// Mitsubishi GX Works2 project: Traffic light_MyTest   PLC: FX3U/FX3UC

PROGRAM MAIN
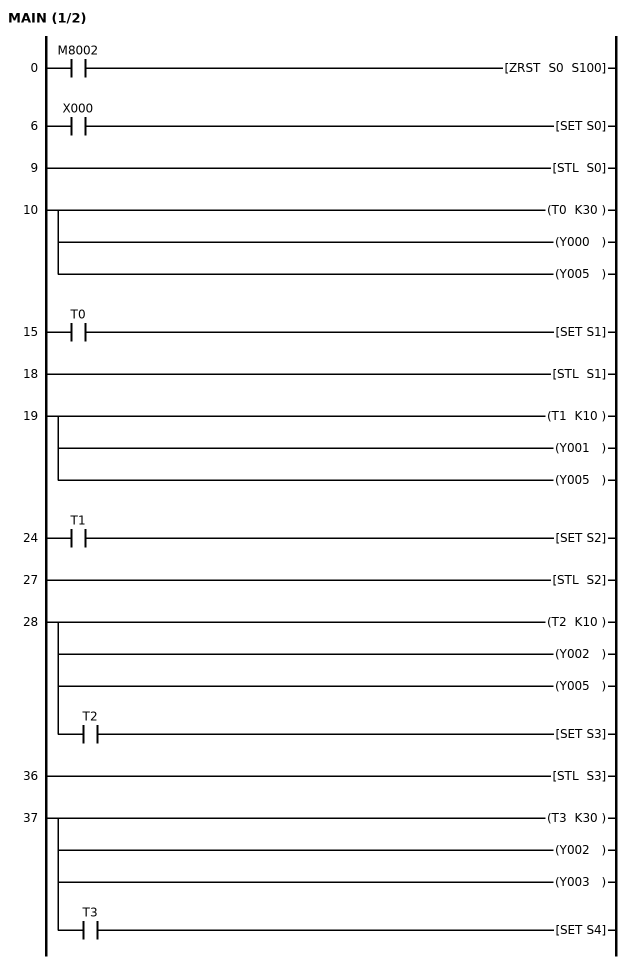
0     LD      M8002
      ZRST    S0 S100
6     LD      X000
      SET     S0
9     STL     S0
10    OUT     T0 K30
      OUT     Y000
      OUT     Y005
15    LD      T0
      SET     S1
18    STL     S1
19    OUT     T1 K10
      OUT     Y001
      OUT     Y005
24    LD      T1
      SET     S2
27    STL     S2
28    OUT     T2 K10
      OUT     Y002
      OUT     Y005
      AND     T2
      SET     S3
36    STL     S3
37    OUT     T3 K30
      OUT     Y002
      OUT     Y003
      AND     T3
      SET     S4
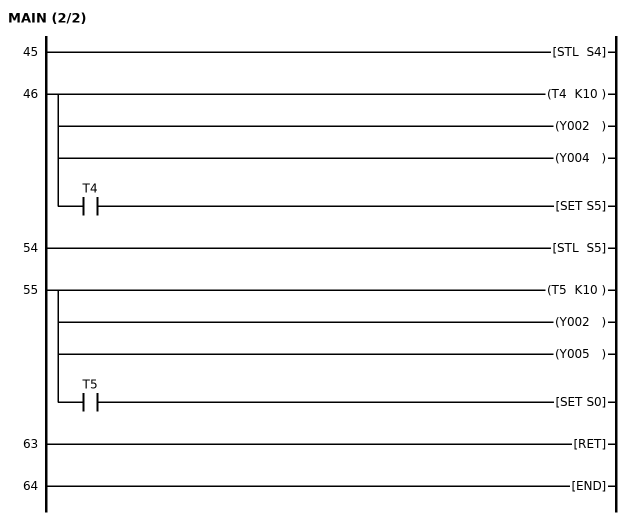
45    STL     S4
46    OUT     T4 K10
      OUT     Y002
      OUT     Y004
      AND     T4
      SET     S5
54    STL     S5
55    OUT     T5 K10
      OUT     Y002
      OUT     Y005
      AND     T5
      SET     S0
63    RET
64    END
END_PROGRAM
